{attribute 'GeneratedUsingTerminal: EK1100-0000-0018'}
{attribute addProperty BoxType "EK1100-0000-0018"}
{attribute addProperty Id "Term_749_EL1809EL1809_32157CFD20Term_750_EL1809EL1809_32157CFD20Term_751_EL1809EL1809_32157CFD20Term_752_EL1809EL1809_32157CFD20Term_753_EL1809EL1809_32157CFD20Term_754_EL1809EL1809_32157CFD20Term_755_EL1809EL1809_32157CFD20Term_756_EL1809EL1809_32157CFD20Term_757_EL1809EL1809_32157CFD20Term_758_EL1809EL1809_32157CFD20Term_759_EL1809EL1809_32157CFD20Term_760_EL1809EL1809_32157CFD20Term_761_EL1809EL1809_32157CFD20Term_762_EL1809EL1809_32157CFD20Term_763_EL1809EL1809_32157CFD20Term_764_EL1809EL1809_32157CFD20Term_765_EL1809EL1809_32157CFD20Term_766_EL1809EL1809_32157CFD20Term_767_EL1809EL1809_32157CFD20Term_768_EL1809EL1809_32157CFD20Term_769_EL1809EL1809_32157CFD20Term_770_EL1809EL1809_32157CFD20Term_771_EL1809EL1809_32157CFD20Term_772_EL1809EL1809_32157CFD20Term_773_EL1809EL1809_32157CFD20Term_774_EL1809EL1809_32157CFD20Term_775_EL1809EL1809_32157CFD20Term_776_EL1809EL1809_32157CFD20Term_777_EL1809EL1809_32157CFD20Term_778_EL1809EL1809_32157CFD20Term_779_EL1809EL1809_32157CFD20Term_780_EL1809EL1809_32157CFD20Term_781_EL1809EL1809_32157CFD20Term_782_EL1809EL1809_32157CFD20Term_783_EL1809EL1809_32157CFD20Term_784_EL1809EL1809_32157CFD20Term_785_EL1809EL1809_32157CFD20Term_786_EL1809EL1809_32157CFD20Term_787_EL1809EL1809_32157CFD20Term_788_EL1809EL1809_32157CFD20Term_789_EL1809EL1809_32157CFD20Term_790_EL1809EL1809_32157CFD20Term_791_EL1809EL1809_32157CFD20Term_792_EL1809EL1809_32157CFD20Term_793_EL1809EL1809_32157CFD20Term_794_EL1809EL1809_32157CFD20Term_795_EL1809EL1809_32157CFD20Term_796_EL1809EL1809_32157CFD20Term_798_EL1809EL1809_32157CFD20Term_799_EL1809EL1809_32157CFD20Term_800_EL1809EL1809_32157CFD20Term_801_EL1809EL1809_32157CFD20Term_802_EL1809EL1809_32157CFD20Term_803_EL1809EL1809_32157CFD20Term_804_EL1809EL1809_32157CFD20Term_805_EL1809EL1809_32157CFD20Term_806_EL1809EL1809_32157CFD20Term_807_EL1809EL1809_32157CFD20Term_808_EL1809EL1809_32157CFD20Term_809_EL1809EL1809_32157CFD20Term_810_EL1809EL1809_32157CFD20Term_811_EL1809EL1809_32157CFD20Term_812_EL1809EL1809_32157CFD20Term_813_EL1809EL1809_32157CFD20Term_814_EL1809EL1809_32157CFD20Term_815_EL1809EL1809_32157CFD20Term_816_EL1809EL1809_32157CFD20Term_817_EL1809EL1809_32157CFD20Term_818_EL1809EL1809_32157CFD20Term_819_EL1809EL1809_32157CFD20Term_820_EL1809EL1809_32157CFD20Term_821_EL1809EL1809_32157CFD20Term_822_EL1809EL1809_32157CFD20Term_823_EL1809EL1809_32157CFD20Term_824_EL1809EL1809_32157CFD20Term_825_EL1809EL1809_32157CFD20Term_826_EL1809EL1809_32157CFD20Term_827_EL1809EL1809_32157CFD20Term_828_EL1809EL1809_32157CFD20Term_859_EL1809EL1809_32157CFD20Term_860_EL1809EL1809_32157CFD20Term_861_EL1809EL1809_32157CFD20Term_862_EL1809EL1809_32157CFD20Term_863_EL1809EL1809_32157CFD20Term_864_EL1809EL1809_32157CFD20Term_865_EL1809EL1809_32157CFD20Term_866_EL1809EL1809_32157CFD20Term_867_EL1809EL1809_32157CFD20Term_868_EL1809EL1809_32157CFD20Term_869_EL1809EL1809_32157CFD20Term_870_EL1809EL1809_32157CFD20Term_871_EL1809EL1809_32157CFD20Term_872_EL1809EL1809_32157CFD20Term_873_EL1809EL1809_32157CFD20Term_874_EL1809EL1809_32157CFD20Term_875_EL1809EL1809_32157CFD20Term_876_EL1809EL1809_32157CFD20Term_877_EL1809EL1809_32157CFD20Term_878_EL1809EL1809_32157CFD20Term_879_EL1809EL1809_32157CFD20Term_880_EK1110EK1110_1FC0878B2"}
{attribute addProperty CRC "3158524849"}
{attribute addProperty Size "2002"}
{attribute addProperty Name "Term 748 (EK1100)"}
TYPE Term_748_EK1100_BC4343B1 EXTENDS EK1100_1FC0878B : 
STRUCT
    {attribute addProperty Name "Term 749 (EL1809)"}
    {attribute addProperty PreviousPort "Term 748 (EK1100) : B"}
    {attribute addProperty SyncUnit "default"}
    Term_749_EL1809 : EL1809_32157CFD;
    {attribute addProperty Name "Term 750 (EL1809)"}
    {attribute addProperty PreviousPort "Term 749 (EL1809) : B"}
    {attribute addProperty SyncUnit "default"}
    Term_750_EL1809 : EL1809_32157CFD;
    {attribute addProperty Name "Term 751 (EL1809)"}
    {attribute addProperty PreviousPort "Term 750 (EL1809) : B"}
    {attribute addProperty SyncUnit "default"}
    Term_751_EL1809 : EL1809_32157CFD;
    {attribute addProperty Name "Term 752 (EL1809)"}
    {attribute addProperty PreviousPort "Term 751 (EL1809) : B"}
    {attribute addProperty SyncUnit "default"}
    Term_752_EL1809 : EL1809_32157CFD;
    {attribute addProperty Name "Term 753 (EL1809)"}
    {attribute addProperty PreviousPort "Term 752 (EL1809) : B"}
    {attribute addProperty SyncUnit "default"}
    Term_753_EL1809 : EL1809_32157CFD;
    {attribute addProperty Name "Term 754 (EL1809)"}
    {attribute addProperty PreviousPort "Term 753 (EL1809) : B"}
    {attribute addProperty SyncUnit "default"}
    Term_754_EL1809 : EL1809_32157CFD;
    {attribute addProperty Name "Term 755 (EL1809)"}
    {attribute addProperty PreviousPort "Term 754 (EL1809) : B"}
    {attribute addProperty SyncUnit "default"}
    Term_755_EL1809 : EL1809_32157CFD;
    {attribute addProperty Name "Term 756 (EL1809)"}
    {attribute addProperty PreviousPort "Term 755 (EL1809) : B"}
    {attribute addProperty SyncUnit "default"}
    Term_756_EL1809 : EL1809_32157CFD;
    {attribute addProperty Name "Term 757 (EL1809)"}
    {attribute addProperty PreviousPort "Term 756 (EL1809) : B"}
    {attribute addProperty SyncUnit "default"}
    Term_757_EL1809 : EL1809_32157CFD;
    {attribute addProperty Name "Term 758 (EL1809)"}
    {attribute addProperty PreviousPort "Term 757 (EL1809) : B"}
    {attribute addProperty SyncUnit "default"}
    Term_758_EL1809 : EL1809_32157CFD;
    {attribute addProperty Name "Term 759 (EL1809)"}
    {attribute addProperty PreviousPort "Term 758 (EL1809) : B"}
    {attribute addProperty SyncUnit "default"}
    Term_759_EL1809 : EL1809_32157CFD;
    {attribute addProperty Name "Term 760 (EL1809)"}
    {attribute addProperty PreviousPort "Term 759 (EL1809) : B"}
    {attribute addProperty SyncUnit "default"}
    Term_760_EL1809 : EL1809_32157CFD;
    {attribute addProperty Name "Term 761 (EL1809)"}
    {attribute addProperty PreviousPort "Term 760 (EL1809) : B"}
    {attribute addProperty SyncUnit "default"}
    Term_761_EL1809 : EL1809_32157CFD;
    {attribute addProperty Name "Term 762 (EL1809)"}
    {attribute addProperty PreviousPort "Term 761 (EL1809) : B"}
    {attribute addProperty SyncUnit "default"}
    Term_762_EL1809 : EL1809_32157CFD;
    {attribute addProperty Name "Term 763 (EL1809)"}
    {attribute addProperty PreviousPort "Term 762 (EL1809) : B"}
    {attribute addProperty SyncUnit "default"}
    Term_763_EL1809 : EL1809_32157CFD;
    {attribute addProperty Name "Term 764 (EL1809)"}
    {attribute addProperty PreviousPort "Term 763 (EL1809) : B"}
    {attribute addProperty SyncUnit "default"}
    Term_764_EL1809 : EL1809_32157CFD;
    {attribute addProperty Name "Term 765 (EL1809)"}
    {attribute addProperty PreviousPort "Term 764 (EL1809) : B"}
    {attribute addProperty SyncUnit "default"}
    Term_765_EL1809 : EL1809_32157CFD;
    {attribute addProperty Name "Term 766 (EL1809)"}
    {attribute addProperty PreviousPort "Term 765 (EL1809) : B"}
    {attribute addProperty SyncUnit "default"}
    Term_766_EL1809 : EL1809_32157CFD;
    {attribute addProperty Name "Term 767 (EL1809)"}
    {attribute addProperty PreviousPort "Term 766 (EL1809) : B"}
    {attribute addProperty SyncUnit "default"}
    Term_767_EL1809 : EL1809_32157CFD;
    {attribute addProperty Name "Term 768 (EL1809)"}
    {attribute addProperty PreviousPort "Term 767 (EL1809) : B"}
    {attribute addProperty SyncUnit "default"}
    Term_768_EL1809 : EL1809_32157CFD;
    {attribute addProperty Name "Term 769 (EL1809)"}
    {attribute addProperty PreviousPort "Term 768 (EL1809) : B"}
    {attribute addProperty SyncUnit "default"}
    Term_769_EL1809 : EL1809_32157CFD;
    {attribute addProperty Name "Term 770 (EL1809)"}
    {attribute addProperty PreviousPort "Term 769 (EL1809) : B"}
    {attribute addProperty SyncUnit "default"}
    Term_770_EL1809 : EL1809_32157CFD;
    {attribute addProperty Name "Term 771 (EL1809)"}
    {attribute addProperty PreviousPort "Term 770 (EL1809) : B"}
    {attribute addProperty SyncUnit "default"}
    Term_771_EL1809 : EL1809_32157CFD;
    {attribute addProperty Name "Term 772 (EL1809)"}
    {attribute addProperty PreviousPort "Term 771 (EL1809) : B"}
    {attribute addProperty SyncUnit "default"}
    Term_772_EL1809 : EL1809_32157CFD;
    {attribute addProperty Name "Term 773 (EL1809)"}
    {attribute addProperty PreviousPort "Term 772 (EL1809) : B"}
    {attribute addProperty SyncUnit "default"}
    Term_773_EL1809 : EL1809_32157CFD;
    {attribute addProperty Name "Term 774 (EL1809)"}
    {attribute addProperty PreviousPort "Term 773 (EL1809) : B"}
    {attribute addProperty SyncUnit "default"}
    Term_774_EL1809 : EL1809_32157CFD;
    {attribute addProperty Name "Term 775 (EL1809)"}
    {attribute addProperty PreviousPort "Term 774 (EL1809) : B"}
    {attribute addProperty SyncUnit "default"}
    Term_775_EL1809 : EL1809_32157CFD;
    {attribute addProperty Name "Term 776 (EL1809)"}
    {attribute addProperty PreviousPort "Term 775 (EL1809) : B"}
    {attribute addProperty SyncUnit "default"}
    Term_776_EL1809 : EL1809_32157CFD;
    {attribute addProperty Name "Term 777 (EL1809)"}
    {attribute addProperty PreviousPort "Term 776 (EL1809) : B"}
    {attribute addProperty SyncUnit "default"}
    Term_777_EL1809 : EL1809_32157CFD;
    {attribute addProperty Name "Term 778 (EL1809)"}
    {attribute addProperty PreviousPort "Term 777 (EL1809) : B"}
    {attribute addProperty SyncUnit "default"}
    Term_778_EL1809 : EL1809_32157CFD;
    {attribute addProperty Name "Term 779 (EL1809)"}
    {attribute addProperty PreviousPort "Term 778 (EL1809) : B"}
    {attribute addProperty SyncUnit "default"}
    Term_779_EL1809 : EL1809_32157CFD;
    {attribute addProperty Name "Term 780 (EL1809)"}
    {attribute addProperty PreviousPort "Term 779 (EL1809) : B"}
    {attribute addProperty SyncUnit "default"}
    Term_780_EL1809 : EL1809_32157CFD;
    {attribute addProperty Name "Term 781 (EL1809)"}
    {attribute addProperty PreviousPort "Term 780 (EL1809) : B"}
    {attribute addProperty SyncUnit "default"}
    Term_781_EL1809 : EL1809_32157CFD;
    {attribute addProperty Name "Term 782 (EL1809)"}
    {attribute addProperty PreviousPort "Term 781 (EL1809) : B"}
    {attribute addProperty SyncUnit "default"}
    Term_782_EL1809 : EL1809_32157CFD;
    {attribute addProperty Name "Term 783 (EL1809)"}
    {attribute addProperty PreviousPort "Term 782 (EL1809) : B"}
    {attribute addProperty SyncUnit "default"}
    Term_783_EL1809 : EL1809_32157CFD;
    {attribute addProperty Name "Term 784 (EL1809)"}
    {attribute addProperty PreviousPort "Term 783 (EL1809) : B"}
    {attribute addProperty SyncUnit "default"}
    Term_784_EL1809 : EL1809_32157CFD;
    {attribute addProperty Name "Term 785 (EL1809)"}
    {attribute addProperty PreviousPort "Term 784 (EL1809) : B"}
    {attribute addProperty SyncUnit "default"}
    Term_785_EL1809 : EL1809_32157CFD;
    {attribute addProperty Name "Term 786 (EL1809)"}
    {attribute addProperty PreviousPort "Term 785 (EL1809) : B"}
    {attribute addProperty SyncUnit "default"}
    Term_786_EL1809 : EL1809_32157CFD;
    {attribute addProperty Name "Term 787 (EL1809)"}
    {attribute addProperty PreviousPort "Term 786 (EL1809) : B"}
    {attribute addProperty SyncUnit "default"}
    Term_787_EL1809 : EL1809_32157CFD;
    {attribute addProperty Name "Term 788 (EL1809)"}
    {attribute addProperty PreviousPort "Term 787 (EL1809) : B"}
    {attribute addProperty SyncUnit "default"}
    Term_788_EL1809 : EL1809_32157CFD;
    {attribute addProperty Name "Term 789 (EL1809)"}
    {attribute addProperty PreviousPort "Term 788 (EL1809) : B"}
    {attribute addProperty SyncUnit "default"}
    Term_789_EL1809 : EL1809_32157CFD;
    {attribute addProperty Name "Term 790 (EL1809)"}
    {attribute addProperty PreviousPort "Term 789 (EL1809) : B"}
    {attribute addProperty SyncUnit "default"}
    Term_790_EL1809 : EL1809_32157CFD;
    {attribute addProperty Name "Term 791 (EL1809)"}
    {attribute addProperty PreviousPort "Term 790 (EL1809) : B"}
    {attribute addProperty SyncUnit "default"}
    Term_791_EL1809 : EL1809_32157CFD;
    {attribute addProperty Name "Term 792 (EL1809)"}
    {attribute addProperty PreviousPort "Term 791 (EL1809) : B"}
    {attribute addProperty SyncUnit "default"}
    Term_792_EL1809 : EL1809_32157CFD;
    {attribute addProperty Name "Term 793 (EL1809)"}
    {attribute addProperty PreviousPort "Term 792 (EL1809) : B"}
    {attribute addProperty SyncUnit "default"}
    Term_793_EL1809 : EL1809_32157CFD;
    {attribute addProperty Name "Term 794 (EL1809)"}
    {attribute addProperty PreviousPort "Term 793 (EL1809) : B"}
    {attribute addProperty SyncUnit "default"}
    Term_794_EL1809 : EL1809_32157CFD;
    {attribute addProperty Name "Term 795 (EL1809)"}
    {attribute addProperty PreviousPort "Term 794 (EL1809) : B"}
    {attribute addProperty SyncUnit "default"}
    Term_795_EL1809 : EL1809_32157CFD;
    {attribute addProperty Name "Term 796 (EL1809)"}
    {attribute addProperty PreviousPort "Term 795 (EL1809) : B"}
    {attribute addProperty SyncUnit "default"}
    Term_796_EL1809 : EL1809_32157CFD;
    {attribute addProperty Name "Term 798 (EL1809)"}
    {attribute addProperty PreviousPort "Term 796 (EL1809) : B"}
    {attribute addProperty SyncUnit "default"}
    Term_798_EL1809 : EL1809_32157CFD;
    {attribute addProperty Name "Term 799 (EL1809)"}
    {attribute addProperty PreviousPort "Term 798 (EL1809) : B"}
    {attribute addProperty SyncUnit "default"}
    Term_799_EL1809 : EL1809_32157CFD;
    {attribute addProperty Name "Term 800 (EL1809)"}
    {attribute addProperty PreviousPort "Term 799 (EL1809) : B"}
    {attribute addProperty SyncUnit "default"}
    Term_800_EL1809 : EL1809_32157CFD;
    {attribute addProperty Name "Term 801 (EL1809)"}
    {attribute addProperty PreviousPort "Term 800 (EL1809) : B"}
    {attribute addProperty SyncUnit "default"}
    Term_801_EL1809 : EL1809_32157CFD;
    {attribute addProperty Name "Term 802 (EL1809)"}
    {attribute addProperty PreviousPort "Term 801 (EL1809) : B"}
    {attribute addProperty SyncUnit "default"}
    Term_802_EL1809 : EL1809_32157CFD;
    {attribute addProperty Name "Term 803 (EL1809)"}
    {attribute addProperty PreviousPort "Term 802 (EL1809) : B"}
    {attribute addProperty SyncUnit "default"}
    Term_803_EL1809 : EL1809_32157CFD;
    {attribute addProperty Name "Term 804 (EL1809)"}
    {attribute addProperty PreviousPort "Term 803 (EL1809) : B"}
    {attribute addProperty SyncUnit "default"}
    Term_804_EL1809 : EL1809_32157CFD;
    {attribute addProperty Name "Term 805 (EL1809)"}
    {attribute addProperty PreviousPort "Term 804 (EL1809) : B"}
    {attribute addProperty SyncUnit "default"}
    Term_805_EL1809 : EL1809_32157CFD;
    {attribute addProperty Name "Term 806 (EL1809)"}
    {attribute addProperty PreviousPort "Term 805 (EL1809) : B"}
    {attribute addProperty SyncUnit "default"}
    Term_806_EL1809 : EL1809_32157CFD;
    {attribute addProperty Name "Term 807 (EL1809)"}
    {attribute addProperty PreviousPort "Term 806 (EL1809) : B"}
    {attribute addProperty SyncUnit "default"}
    Term_807_EL1809 : EL1809_32157CFD;
    {attribute addProperty Name "Term 808 (EL1809)"}
    {attribute addProperty PreviousPort "Term 807 (EL1809) : B"}
    {attribute addProperty SyncUnit "default"}
    Term_808_EL1809 : EL1809_32157CFD;
    {attribute addProperty Name "Term 809 (EL1809)"}
    {attribute addProperty PreviousPort "Term 808 (EL1809) : B"}
    {attribute addProperty SyncUnit "default"}
    Term_809_EL1809 : EL1809_32157CFD;
    {attribute addProperty Name "Term 810 (EL1809)"}
    {attribute addProperty PreviousPort "Term 809 (EL1809) : B"}
    {attribute addProperty SyncUnit "default"}
    Term_810_EL1809 : EL1809_32157CFD;
    {attribute addProperty Name "Term 811 (EL1809)"}
    {attribute addProperty PreviousPort "Term 810 (EL1809) : B"}
    {attribute addProperty SyncUnit "default"}
    Term_811_EL1809 : EL1809_32157CFD;
    {attribute addProperty Name "Term 812 (EL1809)"}
    {attribute addProperty PreviousPort "Term 811 (EL1809) : B"}
    {attribute addProperty SyncUnit "default"}
    Term_812_EL1809 : EL1809_32157CFD;
    {attribute addProperty Name "Term 813 (EL1809)"}
    {attribute addProperty PreviousPort "Term 812 (EL1809) : B"}
    {attribute addProperty SyncUnit "default"}
    Term_813_EL1809 : EL1809_32157CFD;
    {attribute addProperty Name "Term 814 (EL1809)"}
    {attribute addProperty PreviousPort "Term 813 (EL1809) : B"}
    {attribute addProperty SyncUnit "default"}
    Term_814_EL1809 : EL1809_32157CFD;
    {attribute addProperty Name "Term 815 (EL1809)"}
    {attribute addProperty PreviousPort "Term 814 (EL1809) : B"}
    {attribute addProperty SyncUnit "default"}
    Term_815_EL1809 : EL1809_32157CFD;
    {attribute addProperty Name "Term 816 (EL1809)"}
    {attribute addProperty PreviousPort "Term 815 (EL1809) : B"}
    {attribute addProperty SyncUnit "default"}
    Term_816_EL1809 : EL1809_32157CFD;
    {attribute addProperty Name "Term 817 (EL1809)"}
    {attribute addProperty PreviousPort "Term 816 (EL1809) : B"}
    {attribute addProperty SyncUnit "default"}
    Term_817_EL1809 : EL1809_32157CFD;
    {attribute addProperty Name "Term 818 (EL1809)"}
    {attribute addProperty PreviousPort "Term 817 (EL1809) : B"}
    {attribute addProperty SyncUnit "default"}
    Term_818_EL1809 : EL1809_32157CFD;
    {attribute addProperty Name "Term 819 (EL1809)"}
    {attribute addProperty PreviousPort "Term 818 (EL1809) : B"}
    {attribute addProperty SyncUnit "default"}
    Term_819_EL1809 : EL1809_32157CFD;
    {attribute addProperty Name "Term 820 (EL1809)"}
    {attribute addProperty PreviousPort "Term 819 (EL1809) : B"}
    {attribute addProperty SyncUnit "default"}
    Term_820_EL1809 : EL1809_32157CFD;
    {attribute addProperty Name "Term 821 (EL1809)"}
    {attribute addProperty PreviousPort "Term 820 (EL1809) : B"}
    {attribute addProperty SyncUnit "default"}
    Term_821_EL1809 : EL1809_32157CFD;
    {attribute addProperty Name "Term 822 (EL1809)"}
    {attribute addProperty PreviousPort "Term 821 (EL1809) : B"}
    {attribute addProperty SyncUnit "default"}
    Term_822_EL1809 : EL1809_32157CFD;
    {attribute addProperty Name "Term 823 (EL1809)"}
    {attribute addProperty PreviousPort "Term 822 (EL1809) : B"}
    {attribute addProperty SyncUnit "default"}
    Term_823_EL1809 : EL1809_32157CFD;
    {attribute addProperty Name "Term 824 (EL1809)"}
    {attribute addProperty PreviousPort "Term 823 (EL1809) : B"}
    {attribute addProperty SyncUnit "default"}
    Term_824_EL1809 : EL1809_32157CFD;
    {attribute addProperty Name "Term 825 (EL1809)"}
    {attribute addProperty PreviousPort "Term 824 (EL1809) : B"}
    {attribute addProperty SyncUnit "default"}
    Term_825_EL1809 : EL1809_32157CFD;
    {attribute addProperty Name "Term 826 (EL1809)"}
    {attribute addProperty PreviousPort "Term 825 (EL1809) : B"}
    {attribute addProperty SyncUnit "default"}
    Term_826_EL1809 : EL1809_32157CFD;
    {attribute addProperty Name "Term 827 (EL1809)"}
    {attribute addProperty PreviousPort "Term 826 (EL1809) : B"}
    {attribute addProperty SyncUnit "default"}
    Term_827_EL1809 : EL1809_32157CFD;
    {attribute addProperty Name "Term 828 (EL1809)"}
    {attribute addProperty PreviousPort "Term 827 (EL1809) : B"}
    {attribute addProperty SyncUnit "default"}
    Term_828_EL1809 : EL1809_32157CFD;
    {attribute addProperty Name "Term 859 (EL1809)"}
    {attribute addProperty PreviousPort "Term 828 (EL1809) : B"}
    {attribute addProperty SyncUnit "default"}
    Term_859_EL1809 : EL1809_32157CFD;
    {attribute addProperty Name "Term 860 (EL1809)"}
    {attribute addProperty PreviousPort "Term 859 (EL1809) : B"}
    {attribute addProperty SyncUnit "default"}
    Term_860_EL1809 : EL1809_32157CFD;
    {attribute addProperty Name "Term 861 (EL1809)"}
    {attribute addProperty PreviousPort "Term 860 (EL1809) : B"}
    {attribute addProperty SyncUnit "default"}
    Term_861_EL1809 : EL1809_32157CFD;
    {attribute addProperty Name "Term 862 (EL1809)"}
    {attribute addProperty PreviousPort "Term 861 (EL1809) : B"}
    {attribute addProperty SyncUnit "default"}
    Term_862_EL1809 : EL1809_32157CFD;
    {attribute addProperty Name "Term 863 (EL1809)"}
    {attribute addProperty PreviousPort "Term 862 (EL1809) : B"}
    {attribute addProperty SyncUnit "default"}
    Term_863_EL1809 : EL1809_32157CFD;
    {attribute addProperty Name "Term 864 (EL1809)"}
    {attribute addProperty PreviousPort "Term 863 (EL1809) : B"}
    {attribute addProperty SyncUnit "default"}
    Term_864_EL1809 : EL1809_32157CFD;
    {attribute addProperty Name "Term 865 (EL1809)"}
    {attribute addProperty PreviousPort "Term 864 (EL1809) : B"}
    {attribute addProperty SyncUnit "default"}
    Term_865_EL1809 : EL1809_32157CFD;
    {attribute addProperty Name "Term 866 (EL1809)"}
    {attribute addProperty PreviousPort "Term 865 (EL1809) : B"}
    {attribute addProperty SyncUnit "default"}
    Term_866_EL1809 : EL1809_32157CFD;
    {attribute addProperty Name "Term 867 (EL1809)"}
    {attribute addProperty PreviousPort "Term 866 (EL1809) : B"}
    {attribute addProperty SyncUnit "default"}
    Term_867_EL1809 : EL1809_32157CFD;
    {attribute addProperty Name "Term 868 (EL1809)"}
    {attribute addProperty PreviousPort "Term 867 (EL1809) : B"}
    {attribute addProperty SyncUnit "default"}
    Term_868_EL1809 : EL1809_32157CFD;
    {attribute addProperty Name "Term 869 (EL1809)"}
    {attribute addProperty PreviousPort "Term 868 (EL1809) : B"}
    {attribute addProperty SyncUnit "default"}
    Term_869_EL1809 : EL1809_32157CFD;
    {attribute addProperty Name "Term 870 (EL1809)"}
    {attribute addProperty PreviousPort "Term 869 (EL1809) : B"}
    {attribute addProperty SyncUnit "default"}
    Term_870_EL1809 : EL1809_32157CFD;
    {attribute addProperty Name "Term 871 (EL1809)"}
    {attribute addProperty PreviousPort "Term 870 (EL1809) : B"}
    {attribute addProperty SyncUnit "default"}
    Term_871_EL1809 : EL1809_32157CFD;
    {attribute addProperty Name "Term 872 (EL1809)"}
    {attribute addProperty PreviousPort "Term 871 (EL1809) : B"}
    {attribute addProperty SyncUnit "default"}
    Term_872_EL1809 : EL1809_32157CFD;
    {attribute addProperty Name "Term 873 (EL1809)"}
    {attribute addProperty PreviousPort "Term 872 (EL1809) : B"}
    {attribute addProperty SyncUnit "default"}
    Term_873_EL1809 : EL1809_32157CFD;
    {attribute addProperty Name "Term 874 (EL1809)"}
    {attribute addProperty PreviousPort "Term 873 (EL1809) : B"}
    {attribute addProperty SyncUnit "default"}
    Term_874_EL1809 : EL1809_32157CFD;
    {attribute addProperty Name "Term 875 (EL1809)"}
    {attribute addProperty PreviousPort "Term 874 (EL1809) : B"}
    {attribute addProperty SyncUnit "default"}
    Term_875_EL1809 : EL1809_32157CFD;
    {attribute addProperty Name "Term 876 (EL1809)"}
    {attribute addProperty PreviousPort "Term 875 (EL1809) : B"}
    {attribute addProperty SyncUnit "default"}
    Term_876_EL1809 : EL1809_32157CFD;
    {attribute addProperty Name "Term 877 (EL1809)"}
    {attribute addProperty PreviousPort "Term 876 (EL1809) : B"}
    {attribute addProperty SyncUnit "default"}
    Term_877_EL1809 : EL1809_32157CFD;
    {attribute addProperty Name "Term 878 (EL1809)"}
    {attribute addProperty PreviousPort "Term 877 (EL1809) : B"}
    {attribute addProperty SyncUnit "default"}
    Term_878_EL1809 : EL1809_32157CFD;
    {attribute addProperty Name "Term 879 (EL1809)"}
    {attribute addProperty PreviousPort "Term 878 (EL1809) : B"}
    {attribute addProperty SyncUnit "default"}
    Term_879_EL1809 : EL1809_32157CFD;
    {attribute addProperty Name "Term 880 (EK1110)"}
    {attribute addProperty PreviousPort "Term 879 (EL1809) : B"}
    {attribute addProperty SyncUnit "default"}
    Term_880_EK1110 : EK1110_1FC0878B;
END_STRUCT
END_TYPE

(* stored: Version 1.2.0.0, ProductVersion 3.1.4024.11
   DUT Term_748_EK1100_BC4343B1: Id {9d9e8deb-3260-0212-34af-8239b65df1a6} *)
